# EPICS autosave request: iocs/cryo/req/cryo_settings.req
# Operator settings restored across IOC restarts
$(P):TC1:SP
$(P):CMP1:RUN
